FUNCTION_BLOCK FB_AxisStMachineMaster
VAR_IN_OUT
	AxisInOut : AXIS_REF;//AXIS_REF contains input and output
END_VAR
VAR
	nStep : UINT := 10;
	
	fbPower : MC_Power;
		
	errId : UDINT;
	bBusy, bError, bMoveAbs, bMoveVel, bDone, bPower, bReset, bResetDone,bVelocity, bInVelocity, MoveAbsbDone, bDoneHalt, bAborted,bHalt,bHomingDone : BOOL;

	bDemandStop,bDemandVel  AT%I* : BOOL;
	
	fbMoveAbs : MC_MoveAbsolute;
	fTarget	: LREAL := 720;
	fVelocity : LREAL := 36;
	fVelocityInfinite : LREAL := 360;
	fbReset : MC_Reset;//remove error in the NC only for AX8000 but not for AX5000
	fbVelocity : MC_MoveVelocity;
	fbHalt : MC_HALT;
	fbHome : MC_Home;
	bCalibCam AT%I* : BOOL;
	bHome : BOOL;
END_VAR

RunFBs();

CASE nStep OF
	0 : //Idle
		;
	10:
		bPower := TRUE;
		nStep := 15;
	15:
		IF AxisInOut.Status.Error THEN //really at the level of NC
			nStep := 20;
		ELSE
			nstep := 40;
		END_IF
	20:
		bReset := TRUE;
		nstep := 30;	
	30:
		IF bResetDone THEN
			bReset := FALSE;
			nStep := 40;
		END_IF
	40:
		IF fbPower.Status THEN
			bHome := TRUE;
			nStep := 45;
		END_IF
	45:
		IF bHomingDone THEN
			bHome := FALSE;
			nStep := 50;
		END_IF 
	50:
		bMoveAbs := TRUE;
		fTarget	 := 36;//gradi
		fVelocity := 36;
		nstep := 60;
	60:
		IF MoveAbsbDone THEN
			bMoveAbs := FALSE;
			nStep := 65;
		END_IF
	65:
		IF bDemandVel THEN
			nStep := 70;
		END_IF
	70:
		bMoveVel := TRUE;
		fVelocityInfinite := 1440;
		nStep := 80;
	80:
		IF bDemandStop THEN
			bMoveVel := FALSE;
			nStep := 90;
		END_IF
	90:
		bHalt := TRUE;
		nStep := 100;
	
	100:
		IF fbHalt.Done THEN
			bHalt := FALSE;
			nStep := 0;
		END_IF
	ELSE
		;
END_CASE

METHOD RunFBs : BOOL
fbPower(
	Axis:= AxisInOut, 
	Enable:= bPower, 
	Enable_Positive:= TRUE, 
	Enable_Negative:= TRUE, 
	Override:= 100, 
	Busy=>bBusy , 
	Error=>bError, 
	ErrorID=> errId);

fbMoveAbs(
	Axis:= AxisInOut, 
	Execute:= bMoveAbs, 
	Position:= fTarget, 
	Velocity:= fVelocity,  
	Done=> MoveAbsbDone, 
	Busy=>bBusy, 
	Error=>bError, 
	ErrorID=> errId);

fbReset(
	Axis:= AxisInOut, 
	Execute:= bReset, 
	Done=> bResetDone,
	Busy=> bBusy, 
	Error=>bError, 
	ErrorID=>errId);
	
fbVelocity(
	Axis:= AxisInOut, 
	Execute:= bMoveVel, 
	Velocity:= fVelocityInfinite, 
	InVelocity=> bInVelocity, 
	Busy=> bBusy, 
	Error=>bError, 
	ErrorID=>errId);

fbHalt(
	Axis:= AxisInOut, 
	Execute:= bHalt, 
	Done=> bDoneHalt, 
	Busy=> bBusy, 
	CommandAborted=> bAborted, 
	Error=> bError, 
	ErrorID=>errId);

	//without giving special values to the parameters NC parameters are used
fbHome(
	Axis:= AxisInOut, 
	Execute:= bHome, 
	Position:= , 
	HomingMode:= , 
	BufferMode:= , 
	Options:= , 
	bCalibrationCam:= bCalibCam, 
	Done=> bHomingDone, 
	Busy=> , 
	Active=> , 
	CommandAborted=> , 
	Error=> , 
	ErrorID=> );
END_METHOD

END_FUNCTION_BLOCK

(* stored: Version 1.1.0.1, ProductVersion 3.1.4024.13
   POU FB_AxisStMachineMaster: Id {a10afbd2-99b8-4b15-bab4-d05e75652dfb}, SpecialFunc None
   Method RunFBs: Id {06485a6c-8dfd-46c2-924b-ffa80b2f0196} *)
